{attribute 'qualified_only'}
{attribute 'strict'}
TYPE EFeedbackMsgSh10pil :
(
	ShutterIrisPositionMsg := 10
);
END_TYPE

(* stored: Version 1.1.0.1, ProductVersion 3.1.4024.4
   DUT EFeedbackMsgSh10pil: Id {139f0ac4-1e66-4bca-b41b-223b7d530ead} *)
